// SIMATIC S7-200 project (STEP 7-Micro/WIN), CPU 224 REL 02.01

SYMBOL_TABLE USUARIO1
P_MARCHA         I0.0
P_DERECHA        I0.1
P_IZQUIRDA       I0.2
P_PARO           I0.3
BATIDORA         Q0.0
VOLCADO_RECIPIENTE Q0.1
RECOGIDA_RECIPIENTE Q0.2
PISTON           Q0.3
CINTA_DERECHA    Q0.4
CINTA_IZQUIERDA  Q0.5
R_TERMICO        I0.4
END_SYMBOL_TABLE

ORGANIZATION_BLOCK PRINCIPAL:OB1
TITLE=COMENTARIOS DEL PROGRAMA
BEGIN
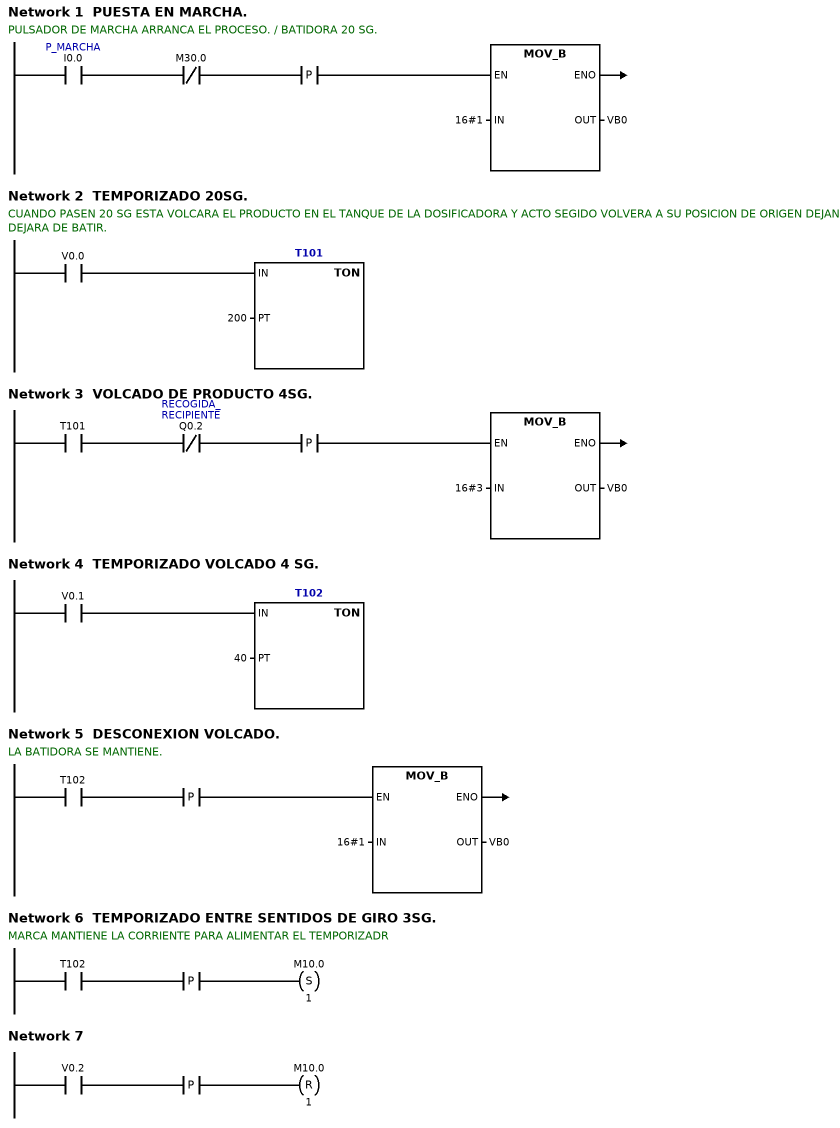
Network 1 // PUESTA EN MARCHA.
// PULSADOR DE MARCHA ARRANCA EL PROCESO.
// BATIDORA 20 SG.
LD     P_MARCHA:I0.0
AN     M30.0
EU
MOVB   16#1, VB0
Network 2 // TEMPORIZADO 20SG.
// CUANDO PASEN 20 SG ESTA VOLCARA EL PRODUCTO EN EL TANQUE DE LA DOSIFICADORA Y ACTO SEGIDO VOLVERA A SU POSICION DE ORIGEN DEJANDO ,MOMENTO ENTONCES QUE LA BATIBORA DEJARA DE BATIR.
LD     V0.0
TON    T101, 200
Network 3 // VOLCADO DE PRODUCTO 4SG.
LD     T101
AN     RECOGIDA_RECIPIENTE:Q0.2
EU
MOVB   16#3, VB0
Network 4 // TEMPORIZADO VOLCADO 4 SG.
LD     V0.1
TON    T102, 40
Network 5 // DESCONEXION VOLCADO.
// LA BATIDORA SE MANTIENE.
LD     T102
EU
MOVB   16#1, VB0
Network 6 // TEMPORIZADO ENTRE SENTIDOS DE GIRO 3SG.
// MARCA MANTIENE LA CORRIENTE PARA ALIMENTAR EL TEMPORIZADR 
LD     T102
EU
S      M10.0, 1
Network 7
LD     V0.2
EU
R      M10.0, 1
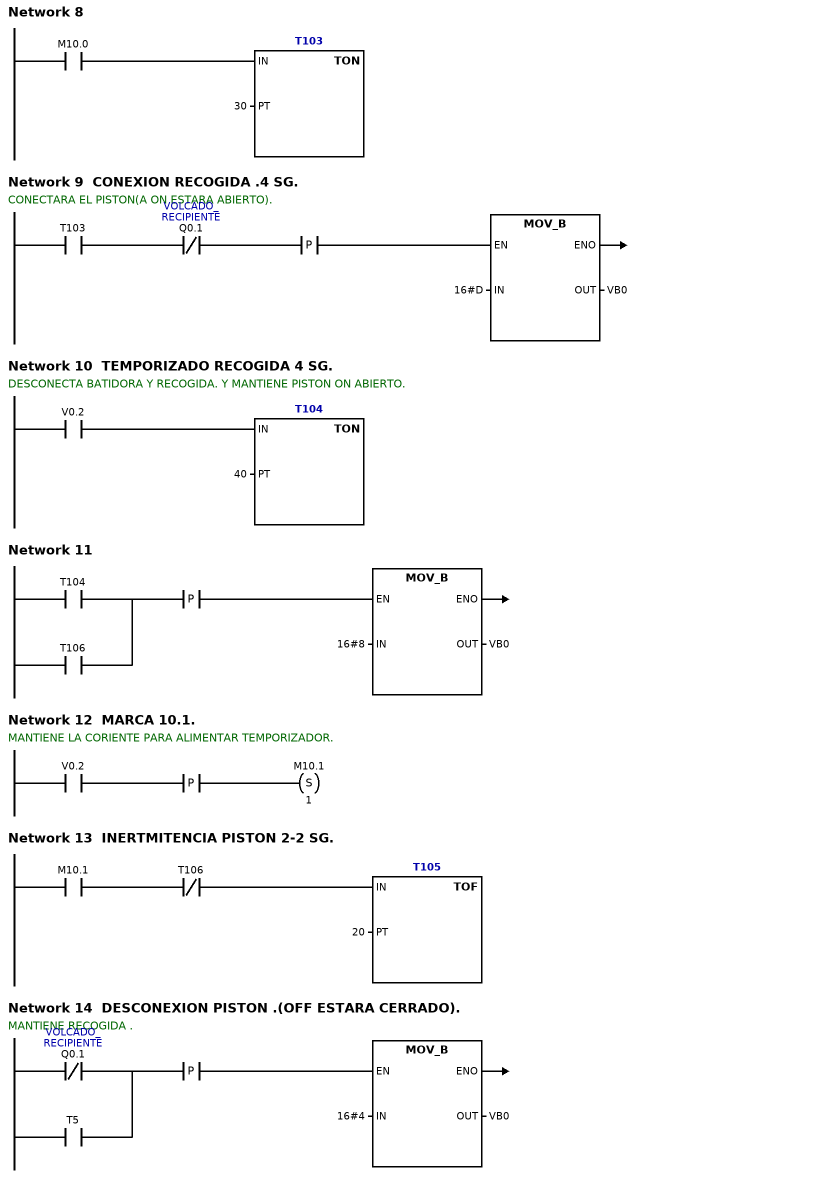
Network 8
LD     M10.0
TON    T103, 30
Network 9 // CONEXION RECOGIDA .4 SG.
// CONECTARA EL PISTON(A ON ESTARA ABIERTO).
LD     T103
AN     VOLCADO_RECIPIENTE:Q0.1
EU
MOVB   16#D, VB0
Network 10 // TEMPORIZADO RECOGIDA 4 SG.
// DESCONECTA BATIDORA Y RECOGIDA. Y MANTIENE PISTON ON ABIERTO.
LD     V0.2
TON    T104, 40
Network 11
LD     T104
O      T106
EU
MOVB   16#8, VB0
Network 12 // MARCA 10.1.
// MANTIENE LA CORIENTE PARA ALIMENTAR TEMPORIZADOR.
LD     V0.2
EU
S      M10.1, 1
Network 13 // INERTMITENCIA PISTON 2-2 SG.
LD     M10.1
AN     T106
TOF    T105, 20
Network 14 // DESCONEXION PISTON .(OFF ESTARA CERRADO).
// MANTIENE RECOGIDA .
LDN    VOLCADO_RECIPIENTE:Q0.1
O      T5
EU
MOVB   16#4, VB0
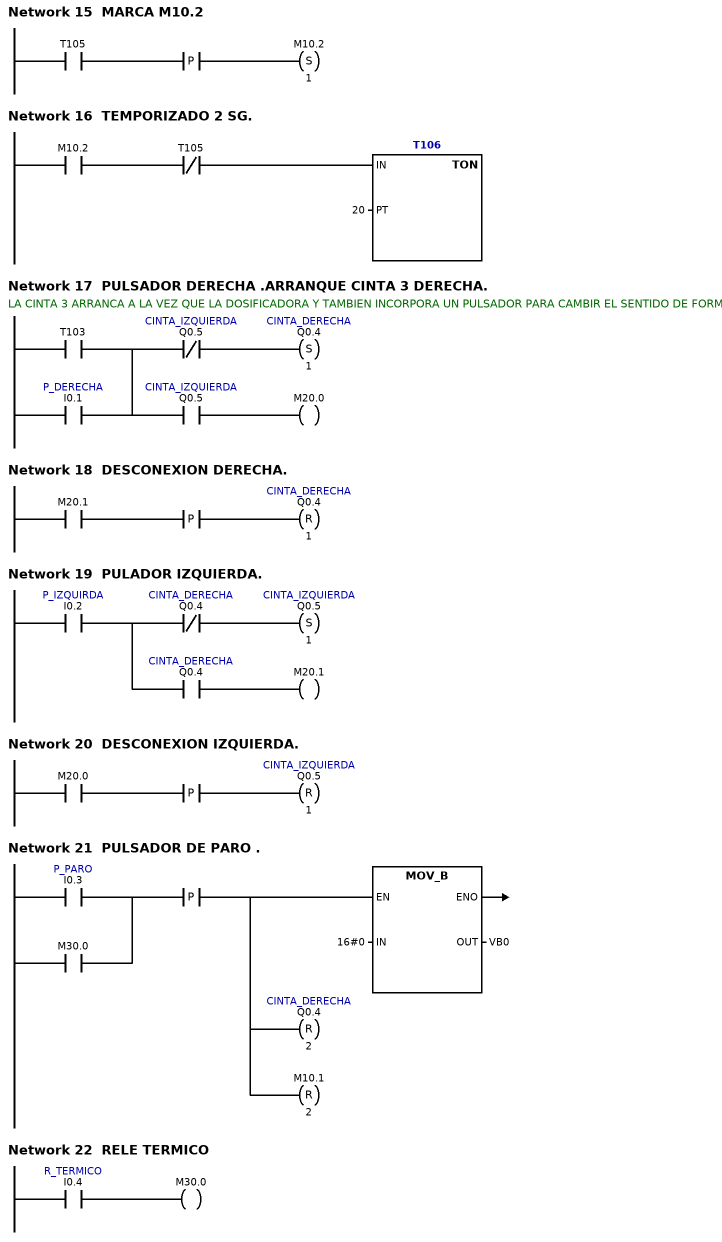
Network 15 // MARCA M10.2
LD     T105
EU
S      M10.2, 1
Network 16 // TEMPORIZADO 2 SG.
LD     M10.2
AN     T105
TON    T106, 20
Network 17 // PULSADOR DERECHA .ARRANQUE CINTA 3 DERECHA.
// LA CINTA 3 ARRANCA A LA VEZ QUE LA DOSIFICADORA Y TAMBIEN INCORPORA UN PULSADOR PARA CAMBIR EL SENTIDO DE FORMA BRUSCA.
LD     T103
O      P_DERECHA:I0.1
LPS
AN     CINTA_IZQUIERDA:Q0.5
S      CINTA_DERECHA:Q0.4, 1
LPP
A      CINTA_IZQUIERDA:Q0.5
=      M20.0
Network 18 // DESCONEXION DERECHA.
LD     M20.1
EU
R      CINTA_DERECHA:Q0.4, 1
Network 19 // PULADOR IZQUIERDA.
LD     P_IZQUIRDA:I0.2
LPS
AN     CINTA_DERECHA:Q0.4
S      CINTA_IZQUIERDA:Q0.5, 1
LPP
A      CINTA_DERECHA:Q0.4
=      M20.1
Network 20 // DESCONEXION IZQUIERDA.
LD     M20.0
EU
R      CINTA_IZQUIERDA:Q0.5, 1
Network 21 // PULSADOR DE PARO .
LD     P_PARO:I0.3
O      M30.0
EU
MOVB   16#0, VB0
R      CINTA_DERECHA:Q0.4, 2
R      M10.1, 2
Network 22 // RELE TERMICO
LD     R_TERMICO:I0.4
=      M30.0
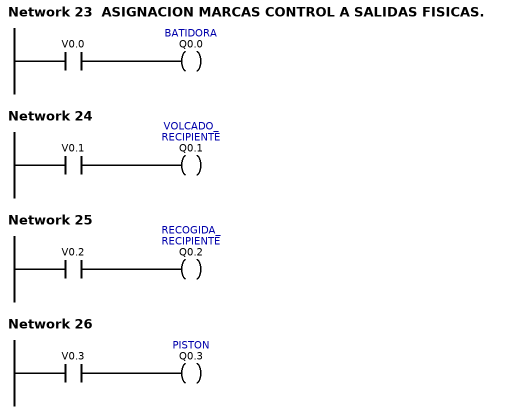
Network 23 // ASIGNACION MARCAS CONTROL A SALIDAS FISICAS.
LD     V0.0
=      BATIDORA:Q0.0
Network 24
LD     V0.1
=      VOLCADO_RECIPIENTE:Q0.1
Network 25
LD     V0.2
=      RECOGIDA_RECIPIENTE:Q0.2
Network 26
LD     V0.3
=      PISTON:Q0.3
END_ORGANIZATION_BLOCK
